{attribute 'qualified_only'}
VAR_GLOBAL
	//Leds
	bLed_Rd1 AT %Q* : BOOL;
	bLed_Rd2 AT %Q* : BOOL;
	bLed_Rd3 AT %Q* : BOOL;
	bLed_Rd4 AT %Q* : BOOL;
	
	bLed_Gn1 AT %Q* : BOOL;
	bLed_Gn2 AT %Q* : BOOL;
	bLed_Gn3 AT %Q* : BOOL;
	bLed_Gn4 AT %Q* : BOOL;
	
	//Buttons
	bButton1 	AT %I* : BOOL;
    bButton2 	AT %I* : BOOL;
    bButton3 	AT %I* : BOOL;
    bButton4 	AT %I* : BOOL;
	bButton5 	AT %I* : BOOL;
    bButton6 	AT %I* : BOOL;
	bHome 		AT %I* : BOOL;
	
	//Sliders
	slider1 : INT;
	slider2 : INT;
	slider3 : INT;
END_VAR

(* stored: Version 1.1.0.1, ProductVersion 3.1.4026.8
   GVL GVL: Id {448d39f8-648e-485a-8da1-4f9a275f6af1} *)
